(* CFC diagram, written out as Structured Text *)
(* KNX Master *)
KNX_master_2(I_Port := IoConfig_Globals.KNX_EIB_TP1_Interface_1, bPortKNX := 2);
STLV80_563.STLV80_A_563_KNX_Card_2_Status := KNX_master_2.sStatus = 'OK';
(* Rom 5H201 *)
(* RB601_V *)
(* RB601_HVAC *)
M2_001_5H201_RB601_V(bPortKNX := 2, dwIndex_DPT := 1, typDPT := typDPT);
STLV80_563.STLV80_A_563_5H201.RB601_V := M2_001_5H201_RB601_V.xSwitch_OUT;
M2_002_5H201_RB601_HVAC(bPortKNX := 2, dwIndex_DPT := 2, typDPT := typDPT);
STLV80_563.STLV80_A_563_5H201.RB601_HVAC := M2_002_5H201_RB601_HVAC.xSwitch_OUT;
(* RT601_CT *)
(* RY601_CV *)
M2_003_5H201_RT601_CT(bPortKNX := 2, dwIndex_DPT := 3, typDPT := typDPT);
STLV80_563.STLV80_A_563_5H201.RT601_CT := M2_003_5H201_RT601_CT.rValue_OUT;
M2_004_5H201_RY601_CV(bPortKNX := 2, dwIndex_DPT := 4, typDPT := typDPT);
STLV80_563.STLV80_A_563_5H201.RY601_CV := M2_004_5H201_RY601_CV.rValue_OUT;
(* LH601_OP *)
(* LH601_CMD *)
M2_005_5H201_LH601_OP(bPortKNX := 2, dwIndex_DPT := 5, rValue_IN := STLV80_563.STLV80_A_563_5H201.LH601_OP, xUpdate_KNX := i = 0, typDPT := typDPT);
M2_006_5H201_LH601_CMD(bPortKNX := 2, dwIndex_DPT := 6, xSwitch_IN := STLV80_563.STLV80_A_563_5H201.LH601_CMD, xUpdate_KNX := i = 1, typDPT := typDPT);
(* LC601_OP *)
(* LC601_CMD *)
M2_007_5H201_LC601_OP(bPortKNX := 2, dwIndex_DPT := 7, rValue_IN := STLV80_563.STLV80_A_563_5H201.LC601_OP, xUpdate_KNX := i = 2, typDPT := typDPT);
M2_008_5H201_LC601_CMD(bPortKNX := 2, dwIndex_DPT := 8, xSwitch_IN := STLV80_563.STLV80_A_563_5H201.LC601_CMD, xUpdate_KNX := i = 3, typDPT := typDPT);
(* RT601_SP *)
(* RT601_SP Feedback *)
M2_009_5H201_RT601_SP(bPortKNX := 2, dwIndex_DPT := 9, rValue_IN := STLV80_563.STLV80_A_563_5H201.RT601_SP_D, xUpdate_KNX := NOT STLV80_563.STLV80_A_563_5H201.RB601_HVAC, typDPT := typDPT);
M2_010_5H201_RT601_SP_FB(bPortKNX := 2, dwIndex_DPT := 10, typDPT := typDPT);
STLV80_563.STLV80_A_563_5H201.RT601_SP_IN := M2_010_5H201_RT601_SP_FB.rValue_OUT;
(* Rom 5I202 *)
(* RB601_V *)
(* RB601_HVAC *)
M2_011_5I202_RB601_V(bPortKNX := 2, dwIndex_DPT := 11, typDPT := typDPT);
STLV80_563.STLV80_A_563_5I202.RB601_V := M2_011_5I202_RB601_V.xSwitch_OUT;
M2_012_5I202_RB601_HVAC(bPortKNX := 2, dwIndex_DPT := 12, typDPT := typDPT);
STLV80_563.STLV80_A_563_5I202.RB601_HVAC := M2_012_5I202_RB601_HVAC.xSwitch_OUT;
(* RT601_CT *)
(* RY601_CV *)
M2_013_5I202_RT601_CT(bPortKNX := 2, dwIndex_DPT := 13, typDPT := typDPT);
STLV80_563.STLV80_A_563_5I202.RT601_CT := M2_013_5I202_RT601_CT.rValue_OUT;
M2_014_5I202_RY601_CV(bPortKNX := 2, dwIndex_DPT := 14, typDPT := typDPT);
STLV80_563.STLV80_A_563_5I202.RY601_CV := M2_014_5I202_RY601_CV.rValue_OUT;
(* LH601_OP *)
(* LH601_CMD *)
M2_015_5I202_LH601_OP(bPortKNX := 2, dwIndex_DPT := 15, rValue_IN := STLV80_563.STLV80_A_563_5I202.LH601_OP, xUpdate_KNX := i = 4, typDPT := typDPT);
M2_016_5I202_LH601_CMD(bPortKNX := 2, dwIndex_DPT := 16, xSwitch_IN := STLV80_563.STLV80_A_563_5I202.LH601_CMD, xUpdate_KNX := i = 5, typDPT := typDPT);
(* LC601_OP *)
(* LC601_CMD *)
M2_017_5I202_LC601_OP(bPortKNX := 2, dwIndex_DPT := 17, rValue_IN := STLV80_563.STLV80_A_563_5I202.LC601_OP, xUpdate_KNX := i = 6, typDPT := typDPT);
M2_018_5I202_LC601_CMD(bPortKNX := 2, dwIndex_DPT := 18, xSwitch_IN := STLV80_563.STLV80_A_563_5I202.LC601_CMD, xUpdate_KNX := i = 7, typDPT := typDPT);
(* RT601_SP *)
(* RT601_SP Feedback *)
M2_019_5I202_RT601_SP(bPortKNX := 2, dwIndex_DPT := 19, rValue_IN := STLV80_563.STLV80_A_563_5I202.RT601_SP_D, xUpdate_KNX := NOT STLV80_563.STLV80_A_563_5I202.RB601_HVAC, typDPT := typDPT);
M2_020_5I202_RT601_SP_FB(bPortKNX := 2, dwIndex_DPT := 20, typDPT := typDPT);
STLV80_563.STLV80_A_563_5I202.RT601_SP_IN := M2_020_5I202_RT601_SP_FB.rValue_OUT;
(* Rom 5I301 *)
(* RB601_V *)
(* RB601_HVAC *)
M2_021_5I301_RB601_V(bPortKNX := 2, dwIndex_DPT := 21, typDPT := typDPT);
STLV80_563.STLV80_A_563_5I301.RB601_V := M2_021_5I301_RB601_V.xSwitch_OUT;
M2_022_5I301_RB601_HVAC(bPortKNX := 2, dwIndex_DPT := 22, typDPT := typDPT);
STLV80_563.STLV80_A_563_5I301.RB601_HVAC := M2_022_5I301_RB601_HVAC.xSwitch_OUT;
(* RT601_CT *)
(* RY601_CV *)
M2_023_5I301_RT601_CT(bPortKNX := 2, dwIndex_DPT := 23, typDPT := typDPT);
STLV80_563.STLV80_A_563_5I301.RT601_CT := M2_023_5I301_RT601_CT.rValue_OUT;
M2_024_5I301_RY601_CV(bPortKNX := 2, dwIndex_DPT := 24, typDPT := typDPT);
STLV80_563.STLV80_A_563_5I301.RY601_CV := M2_024_5I301_RY601_CV.rValue_OUT;
(* LH601_OP *)
(* LH601_CMD *)
M2_025_5I301_LH601_OP(bPortKNX := 2, dwIndex_DPT := 25, rValue_IN := STLV80_563.STLV80_A_563_5I301.LH601_OP, xUpdate_KNX := i = 8, typDPT := typDPT);
M2_026_5I301_LH601_CMD(bPortKNX := 2, dwIndex_DPT := 26, xSwitch_IN := STLV80_563.STLV80_A_563_5I301.LH601_CMD, xUpdate_KNX := i = 9, typDPT := typDPT);
(* LC601_OP *)
(* LC601_CMD *)
M2_027_5I301_LC601_OP(bPortKNX := 2, dwIndex_DPT := 27, rValue_IN := STLV80_563.STLV80_A_563_5I301.LC601_OP, xUpdate_KNX := i = 10, typDPT := typDPT);
M2_028_5I301_LC601_CMD(bPortKNX := 2, dwIndex_DPT := 28, xSwitch_IN := STLV80_563.STLV80_A_563_5I301.LC601_CMD, xUpdate_KNX := i = 11, typDPT := typDPT);
(* RT601_SP *)
(* RT601_SP Feedback *)
M2_029_5I301_RT601_SP(bPortKNX := 2, dwIndex_DPT := 29, rValue_IN := STLV80_563.STLV80_A_563_5I301.RT601_SP_D, xUpdate_KNX := NOT STLV80_563.STLV80_A_563_5I301.RB601_HVAC, typDPT := typDPT);
M2_030_5I301_RT601_SP_FB(bPortKNX := 2, dwIndex_DPT := 30, typDPT := typDPT);
STLV80_563.STLV80_A_563_5I301.RT601_SP_IN := M2_030_5I301_RT601_SP_FB.rValue_OUT;
(* Rom 5I302 *)
(* RB601_V *)
(* RB601_HVAC *)
M2_031_5I302_RB601_V(bPortKNX := 2, dwIndex_DPT := 31, typDPT := typDPT);
STLV80_563.STLV80_A_563_5I302.RB601_V := M2_031_5I302_RB601_V.xSwitch_OUT;
M2_032_5I302_RB601_HVAC(bPortKNX := 2, dwIndex_DPT := 32, typDPT := typDPT);
STLV80_563.STLV80_A_563_5I302.RB601_HVAC := M2_032_5I302_RB601_HVAC.xSwitch_OUT;
(* RT601_CT *)
(* RY601_CV *)
M2_033_5I302_RT601_CT(bPortKNX := 2, dwIndex_DPT := 33, typDPT := typDPT);
STLV80_563.STLV80_A_563_5I302.RT601_CT := M2_033_5I302_RT601_CT.rValue_OUT;
M2_034_5I302_RY601_CV(bPortKNX := 2, dwIndex_DPT := 34, typDPT := typDPT);
STLV80_563.STLV80_A_563_5I302.RY601_CV := M2_034_5I302_RY601_CV.rValue_OUT;
(* LH601_OP *)
(* LH601_CMD *)
M2_035_5I302_LH601_OP(bPortKNX := 2, dwIndex_DPT := 35, rValue_IN := STLV80_563.STLV80_A_563_5I302.LH601_OP, xUpdate_KNX := i = 12, typDPT := typDPT);
M2_036_5I302_LH601_CMD(bPortKNX := 2, dwIndex_DPT := 36, xSwitch_IN := STLV80_563.STLV80_A_563_5I302.LH601_CMD, xUpdate_KNX := i = 13, typDPT := typDPT);
(* LC601_OP *)
(* LC601_CMD *)
M2_037_5I302_LC601_OP(bPortKNX := 2, dwIndex_DPT := 37, rValue_IN := STLV80_563.STLV80_A_563_5I302.LC601_OP, xUpdate_KNX := i = 14, typDPT := typDPT);
M2_038_5I302_LC601_CMD(bPortKNX := 2, dwIndex_DPT := 38, xSwitch_IN := STLV80_563.STLV80_A_563_5I302.LC601_CMD, xUpdate_KNX := i = 15, typDPT := typDPT);
(* RT601_SP *)
(* RT601_SP Feedback *)
M2_039_5I302_RT601_SP(bPortKNX := 2, dwIndex_DPT := 39, rValue_IN := STLV80_563.STLV80_A_563_5I302.RT601_SP_D, xUpdate_KNX := NOT STLV80_563.STLV80_A_563_5I302.RB601_HVAC, typDPT := typDPT);
M2_040_5I302_RT601_SP_FB(bPortKNX := 2, dwIndex_DPT := 40, typDPT := typDPT);
STLV80_563.STLV80_A_563_5I302.RT601_SP_IN := M2_040_5I302_RT601_SP_FB.rValue_OUT;
(* Rom 5J201 *)
(* RB601_V *)
(* RB601_HVAC *)
M2_041_5J201_RB601_V(bPortKNX := 2, dwIndex_DPT := 41, typDPT := typDPT);
STLV80_563.STLV80_A_563_5J201.RB601_V := M2_041_5J201_RB601_V.xSwitch_OUT;
M2_042_5J201_RB601_HVAC(bPortKNX := 2, dwIndex_DPT := 42, typDPT := typDPT);
STLV80_563.STLV80_A_563_5J201.RB601_HVAC := M2_042_5J201_RB601_HVAC.xSwitch_OUT;
(* RT601_CT *)
(* RY601_CV *)
M2_043_5J201_RT601_CT(bPortKNX := 2, dwIndex_DPT := 43, typDPT := typDPT);
STLV80_563.STLV80_A_563_5J201.RT601_CT := M2_043_5J201_RT601_CT.rValue_OUT;
M2_044_5J201_RY601_CV(bPortKNX := 2, dwIndex_DPT := 44, typDPT := typDPT);
STLV80_563.STLV80_A_563_5J201.RY601_CV := M2_044_5J201_RY601_CV.rValue_OUT;
(* LH601_OP *)
(* LH601_CMD *)
M2_045_5J201_LH601_OP(bPortKNX := 2, dwIndex_DPT := 45, rValue_IN := STLV80_563.STLV80_A_563_5J201.LH601_OP, xUpdate_KNX := i = 16, typDPT := typDPT);
M2_046_5J201_LH601_CMD(bPortKNX := 2, dwIndex_DPT := 46, xSwitch_IN := STLV80_563.STLV80_A_563_5J201.LH601_CMD, xUpdate_KNX := i = 17, typDPT := typDPT);
(* LC601_OP *)
(* LC601_CMD *)
M2_047_5J201_LC601_OP(bPortKNX := 2, dwIndex_DPT := 47, rValue_IN := STLV80_563.STLV80_A_563_5J201.LC601_OP, xUpdate_KNX := i = 18, typDPT := typDPT);
M2_048_5J201_LC601_CMD(bPortKNX := 2, dwIndex_DPT := 48, xSwitch_IN := STLV80_563.STLV80_A_563_5J201.LC601_CMD, xUpdate_KNX := i = 19, typDPT := typDPT);
(* RT601_SP *)
(* RT601_SP Feedback *)
M2_049_5J201_RT601_SP(bPortKNX := 2, dwIndex_DPT := 49, rValue_IN := STLV80_563.STLV80_A_563_5J201.RT601_SP_D, xUpdate_KNX := NOT STLV80_563.STLV80_A_563_5J201.RB601_HVAC, typDPT := typDPT);
M2_050_5J201_RT601_SP_FB(bPortKNX := 2, dwIndex_DPT := 50, typDPT := typDPT);
STLV80_563.STLV80_A_563_5J201.RT601_SP_IN := M2_050_5J201_RT601_SP_FB.rValue_OUT;
(* Rom 5J202 *)
(* RB601_V *)
(* RB601_HVAC *)
M2_051_5J202_RB601_V(bPortKNX := 2, dwIndex_DPT := 51, typDPT := typDPT);
STLV80_563.STLV80_A_563_5J202.RB601_V := M2_051_5J202_RB601_V.xSwitch_OUT;
M2_052_5J202_RB601_HVAC(bPortKNX := 2, dwIndex_DPT := 52, typDPT := typDPT);
STLV80_563.STLV80_A_563_5J202.RB601_HVAC := M2_052_5J202_RB601_HVAC.xSwitch_OUT;
(* RT601_CT *)
(* RY601_CV *)
M2_053_5J202_RT601_CT(bPortKNX := 2, dwIndex_DPT := 53, typDPT := typDPT);
STLV80_563.STLV80_A_563_5J202.RT601_CT := M2_053_5J202_RT601_CT.rValue_OUT;
M2_054_5J202_RY601_CV(bPortKNX := 2, dwIndex_DPT := 54, typDPT := typDPT);
STLV80_563.STLV80_A_563_5J202.RY601_CV := M2_054_5J202_RY601_CV.rValue_OUT;
(* LH601_OP *)
(* LH601_CMD *)
M2_055_5J202_LH601_OP(bPortKNX := 2, dwIndex_DPT := 55, rValue_IN := STLV80_563.STLV80_A_563_5J202.LH601_OP, xUpdate_KNX := i = 20, typDPT := typDPT);
M2_056_5J202_LH601_CMD(bPortKNX := 2, dwIndex_DPT := 56, xSwitch_IN := STLV80_563.STLV80_A_563_5J202.LH601_CMD, xUpdate_KNX := i = 21, typDPT := typDPT);
(* LC601_OP *)
(* LC601_CMD *)
M2_057_5J202_LC601_OP(bPortKNX := 2, dwIndex_DPT := 57, rValue_IN := STLV80_563.STLV80_A_563_5J202.LC601_OP, xUpdate_KNX := i = 22, typDPT := typDPT);
M2_058_5J202_LC601_CMD(bPortKNX := 2, dwIndex_DPT := 58, xSwitch_IN := STLV80_563.STLV80_A_563_5J202.LC601_CMD, xUpdate_KNX := i = 23, typDPT := typDPT);
(* RT601_SP *)
(* RT601_SP Feedback *)
M2_059_5J202_RT601_SP(bPortKNX := 2, dwIndex_DPT := 59, rValue_IN := STLV80_563.STLV80_A_563_5J202.RT601_SP_D, xUpdate_KNX := NOT STLV80_563.STLV80_A_563_5J202.RB601_HVAC, typDPT := typDPT);
M2_060_5J202_RT601_SP_FB(bPortKNX := 2, dwIndex_DPT := 60, typDPT := typDPT);
STLV80_563.STLV80_A_563_5J202.RT601_SP_IN := M2_060_5J202_RT601_SP_FB.rValue_OUT;
(* Rom 5J301 *)
(* RB601_V *)
(* RB601_HVAC *)
M2_061_5J301_RB601_V(bPortKNX := 2, dwIndex_DPT := 61, typDPT := typDPT);
STLV80_563.STLV80_A_563_5J301.RB601_V := M2_061_5J301_RB601_V.xSwitch_OUT;
M2_062_5J301_RB601_HVAC(bPortKNX := 2, dwIndex_DPT := 62, typDPT := typDPT);
STLV80_563.STLV80_A_563_5J301.RB601_HVAC := M2_062_5J301_RB601_HVAC.xSwitch_OUT;
(* RT601_CT *)
(* RY601_CV *)
M2_063_5J301_RT601_CT(bPortKNX := 2, dwIndex_DPT := 63, typDPT := typDPT);
STLV80_563.STLV80_A_563_5J301.RT601_CT := M2_063_5J301_RT601_CT.rValue_OUT;
M2_064_5J301_RY601_CV(bPortKNX := 2, dwIndex_DPT := 64, typDPT := typDPT);
STLV80_563.STLV80_A_563_5J301.RY601_CV := M2_064_5J301_RY601_CV.rValue_OUT;
(* LH601_OP *)
(* LH601_CMD *)
M2_065_5J301_LH601_OP(bPortKNX := 2, dwIndex_DPT := 65, rValue_IN := STLV80_563.STLV80_A_563_5J301.LH601_OP, xUpdate_KNX := i = 24, typDPT := typDPT);
M2_066_5J301_LH601_CMD(bPortKNX := 2, dwIndex_DPT := 66, xSwitch_IN := STLV80_563.STLV80_A_563_5J301.LH601_CMD, xUpdate_KNX := i = 25, typDPT := typDPT);
(* LC601_OP *)
(* LC601_CMD *)
M2_067_5J301_LC601_OP(bPortKNX := 2, dwIndex_DPT := 67, rValue_IN := STLV80_563.STLV80_A_563_5J301.LC601_OP, xUpdate_KNX := i = 26, typDPT := typDPT);
M2_068_5J301_LC601_CMD(bPortKNX := 2, dwIndex_DPT := 68, xSwitch_IN := STLV80_563.STLV80_A_563_5J301.LC601_CMD, xUpdate_KNX := i = 27, typDPT := typDPT);
(* RT601_SP *)
(* RT601_SP Feedback *)
M2_069_5J301_RT601_SP(bPortKNX := 2, dwIndex_DPT := 69, rValue_IN := STLV80_563.STLV80_A_563_5J301.RT601_SP_D, xUpdate_KNX := NOT STLV80_563.STLV80_A_563_5J301.RB601_HVAC, typDPT := typDPT);
M2_070_5J301_RT601_SP_FB(bPortKNX := 2, dwIndex_DPT := 70, typDPT := typDPT);
STLV80_563.STLV80_A_563_5J301.RT601_SP_IN := M2_070_5J301_RT601_SP_FB.rValue_OUT;
(* Rom 5K302 *)
(* RB601_V *)
(* RB601_HVAC *)
M2_071_5K302_RB601_V(bPortKNX := 2, dwIndex_DPT := 71, typDPT := typDPT);
STLV80_563.STLV80_A_563_5K302.RB601_V := M2_071_5K302_RB601_V.xSwitch_OUT;
M2_072_5K302_RB601_HVAC(bPortKNX := 2, dwIndex_DPT := 72, typDPT := typDPT);
STLV80_563.STLV80_A_563_5K302.RB601_HVAC := M2_072_5K302_RB601_HVAC.xSwitch_OUT;
(* RT601_CT *)
(* RY601_CV *)
M2_073_5K302_RT601_CT(bPortKNX := 2, dwIndex_DPT := 73, typDPT := typDPT);
STLV80_563.STLV80_A_563_5K302.RT601_CT := M2_073_5K302_RT601_CT.rValue_OUT;
M2_074_5K302_RY601_CV(bPortKNX := 2, dwIndex_DPT := 74, typDPT := typDPT);
STLV80_563.STLV80_A_563_5K302.RY601_CV := M2_074_5K302_RY601_CV.rValue_OUT;
(* LH601_OP *)
(* LH601_CMD *)
M2_075_5K302_LH601_OP(bPortKNX := 2, dwIndex_DPT := 75, rValue_IN := STLV80_563.STLV80_A_563_5K302.LH601_OP, xUpdate_KNX := i = 28, typDPT := typDPT);
M2_076_5K302_LH601_CMD(bPortKNX := 2, dwIndex_DPT := 76, xSwitch_IN := STLV80_563.STLV80_A_563_5K302.LH601_CMD, xUpdate_KNX := i = 29, typDPT := typDPT);
(* LC601_OP *)
(* LC601_CMD *)
M2_077_5K302_LC601_OP(bPortKNX := 2, dwIndex_DPT := 77, rValue_IN := STLV80_563.STLV80_A_563_5K302.LC601_OP, xUpdate_KNX := i = 30, typDPT := typDPT);
M2_078_5K302_LC601_CMD(bPortKNX := 2, dwIndex_DPT := 78, xSwitch_IN := STLV80_563.STLV80_A_563_5K302.LC601_CMD, xUpdate_KNX := i = 31, typDPT := typDPT);
(* RT601_SP *)
(* RT601_SP Feedback *)
M2_079_5K302_RT601_SP(bPortKNX := 2, dwIndex_DPT := 79, rValue_IN := STLV80_563.STLV80_A_563_5K302.RT601_SP_D, xUpdate_KNX := NOT STLV80_563.STLV80_A_563_5K302.RB601_HVAC, typDPT := typDPT);
M2_080_5K302_RT601_SP_FB(bPortKNX := 2, dwIndex_DPT := 80, typDPT := typDPT);
STLV80_563.STLV80_A_563_5K302.RT601_SP_IN := M2_080_5K302_RT601_SP_FB.rValue_OUT;
(* Rom 5K201 *)
(* RB601_V *)
(* RB601_HVAC *)
M2_081_5K201_RB601_V(bPortKNX := 2, dwIndex_DPT := 81, typDPT := typDPT);
STLV80_563.STLV80_A_563_5K201.RB601_V := M2_081_5K201_RB601_V.xSwitch_OUT;
M2_082_5K201_RB601_HVAC(bPortKNX := 2, dwIndex_DPT := 82, typDPT := typDPT);
STLV80_563.STLV80_A_563_5K201.RB601_HVAC := M2_082_5K201_RB601_HVAC.xSwitch_OUT;
(* RT601_CT *)
(* RY601_CV *)
M2_083_5K201_RT601_CT(bPortKNX := 2, dwIndex_DPT := 83, typDPT := typDPT);
STLV80_563.STLV80_A_563_5K201.RT601_CT := M2_083_5K201_RT601_CT.rValue_OUT;
M2_084_5K201_RY601_CV(bPortKNX := 2, dwIndex_DPT := 84, typDPT := typDPT);
STLV80_563.STLV80_A_563_5K201.RY601_CV := M2_084_5K201_RY601_CV.rValue_OUT;
(* LH601_OP *)
(* LH601_CMD *)
M2_085_5K201_LH601_OP(bPortKNX := 2, dwIndex_DPT := 85, rValue_IN := STLV80_563.STLV80_A_563_5K201.LH601_OP, xUpdate_KNX := i = 32, typDPT := typDPT);
M2_086_5K201_LH601_CMD(bPortKNX := 2, dwIndex_DPT := 86, xSwitch_IN := STLV80_563.STLV80_A_563_5K201.LH601_CMD, xUpdate_KNX := i = 33, typDPT := typDPT);
(* LC601_OP *)
(* LC601_CMD *)
M2_087_5K201_LC601_OP(bPortKNX := 2, dwIndex_DPT := 87, rValue_IN := STLV80_563.STLV80_A_563_5K201.LC601_OP, xUpdate_KNX := i = 34, typDPT := typDPT);
M2_088_5K201_LC601_CMD(bPortKNX := 2, dwIndex_DPT := 88, xSwitch_IN := STLV80_563.STLV80_A_563_5K201.LC601_CMD, xUpdate_KNX := i = 35, typDPT := typDPT);
(* RT601_SP *)
(* RT601_SP Feedback *)
M2_089_5K201_RT601_SP(bPortKNX := 2, dwIndex_DPT := 89, rValue_IN := STLV80_563.STLV80_A_563_5K201.RT601_SP_D, xUpdate_KNX := NOT STLV80_563.STLV80_A_563_5K201.RB601_HVAC, typDPT := typDPT);
M2_090_5K201_RT601_SP_FB(bPortKNX := 2, dwIndex_DPT := 90, typDPT := typDPT);
STLV80_563.STLV80_A_563_5K201.RT601_SP_IN := M2_090_5K201_RT601_SP_FB.rValue_OUT;
(* Rom 5K202 *)
(* RB601_V *)
(* RB601_HVAC *)
M2_091_5K202_RB601_V(bPortKNX := 2, dwIndex_DPT := 91, typDPT := typDPT);
STLV80_563.STLV80_A_563_5K202.RB601_V := M2_091_5K202_RB601_V.xSwitch_OUT;
M2_092_5K202_RB601_HVAC(bPortKNX := 2, dwIndex_DPT := 92, typDPT := typDPT);
STLV80_563.STLV80_A_563_5K202.RB601_HVAC := M2_092_5K202_RB601_HVAC.xSwitch_OUT;
(* RT601_CT *)
(* RY601_CV *)
M2_093_5K202_RT601_CT(bPortKNX := 2, dwIndex_DPT := 93, typDPT := typDPT);
STLV80_563.STLV80_A_563_5K202.RT601_CT := M2_093_5K202_RT601_CT.rValue_OUT;
M2_094_5K202_RY601_CV(bPortKNX := 2, dwIndex_DPT := 94, typDPT := typDPT);
STLV80_563.STLV80_A_563_5K202.RY601_CV := M2_094_5K202_RY601_CV.rValue_OUT;
(* LH601_OP *)
(* LH601_CMD *)
M2_095_5K202_LH601_OP(bPortKNX := 2, dwIndex_DPT := 95, rValue_IN := STLV80_563.STLV80_A_563_5K202.LH601_OP, xUpdate_KNX := i = 36, typDPT := typDPT);
M2_096_5K202_LH601_CMD(bPortKNX := 2, dwIndex_DPT := 96, xSwitch_IN := STLV80_563.STLV80_A_563_5K202.LH601_CMD, xUpdate_KNX := i = 37, typDPT := typDPT);
(* LC601_OP *)
(* LC601_CMD *)
M2_097_5K202_LC601_OP(bPortKNX := 2, dwIndex_DPT := 97, rValue_IN := STLV80_563.STLV80_A_563_5K202.LC601_OP, xUpdate_KNX := i = 38, typDPT := typDPT);
M2_098_5K202_LC601_CMD(bPortKNX := 2, dwIndex_DPT := 98, xSwitch_IN := STLV80_563.STLV80_A_563_5K202.LC601_CMD, xUpdate_KNX := i = 39, typDPT := typDPT);
(* RT601_SP *)
(* RT601_SP Feedback *)
M2_099_5K202_RT601_SP(bPortKNX := 2, dwIndex_DPT := 99, rValue_IN := STLV80_563.STLV80_A_563_5K202.RT601_SP_D, xUpdate_KNX := NOT STLV80_563.STLV80_A_563_5K202.RB601_HVAC, typDPT := typDPT);
M2_100_5K202_RT601_SP_FB(bPortKNX := 2, dwIndex_DPT := 100, typDPT := typDPT);
STLV80_563.STLV80_A_563_5K202.RT601_SP_IN := M2_100_5K202_RT601_SP_FB.rValue_OUT;
(* Rom 5K301 *)
(* RB601_V *)
(* RB601_HVAC *)
M2_101_5K301_RB601_V(bPortKNX := 2, dwIndex_DPT := 101, typDPT := typDPT);
STLV80_563.STLV80_A_563_5K301.RB601_V := M2_101_5K301_RB601_V.xSwitch_OUT;
M2_102_5K301_RB601_HVAC(bPortKNX := 2, dwIndex_DPT := 102, typDPT := typDPT);
STLV80_563.STLV80_A_563_5K301.RB601_HVAC := M2_102_5K301_RB601_HVAC.xSwitch_OUT;
(* RT601_CT *)
(* RY601_CV *)
M2_103_5K301_RT601_CT(bPortKNX := 2, dwIndex_DPT := 103, typDPT := typDPT);
STLV80_563.STLV80_A_563_5K301.RT601_CT := M2_103_5K301_RT601_CT.rValue_OUT;
M2_104_5K301_RY601_CV(bPortKNX := 2, dwIndex_DPT := 104, typDPT := typDPT);
STLV80_563.STLV80_A_563_5K301.RY601_CV := M2_104_5K301_RY601_CV.rValue_OUT;
(* LH601_OP *)
(* LH601_CMD *)
M2_105_5K301_LH601_OP(bPortKNX := 2, dwIndex_DPT := 105, rValue_IN := STLV80_563.STLV80_A_563_5K301.LH601_OP, xUpdate_KNX := i = 40, typDPT := typDPT);
M2_106_5K301_LH601_CMD(bPortKNX := 2, dwIndex_DPT := 106, xSwitch_IN := STLV80_563.STLV80_A_563_5K301.LH601_CMD, xUpdate_KNX := i = 41, typDPT := typDPT);
(* LC601_OP *)
(* LC601_CMD *)
M2_107_5K301_LC601_OP(bPortKNX := 2, dwIndex_DPT := 107, rValue_IN := STLV80_563.STLV80_A_563_5K301.LC601_OP, xUpdate_KNX := i = 42, typDPT := typDPT);
M2_108_5K301_LC601_CMD(bPortKNX := 2, dwIndex_DPT := 108, xSwitch_IN := STLV80_563.STLV80_A_563_5K301.LC601_CMD, xUpdate_KNX := i = 43, typDPT := typDPT);
(* RT601_SP *)
(* RT601_SP Feedback *)
M2_109_5K301_RT601_SP(bPortKNX := 2, dwIndex_DPT := 109, rValue_IN := STLV80_563.STLV80_A_563_5K301.RT601_SP_D, xUpdate_KNX := NOT STLV80_563.STLV80_A_563_5K301.RB601_HVAC, typDPT := typDPT);
M2_110_5K301_RT601_SP_FB(bPortKNX := 2, dwIndex_DPT := 110, typDPT := typDPT);
STLV80_563.STLV80_A_563_5K301.RT601_SP_IN := M2_110_5K301_RT601_SP_FB.rValue_OUT;
(* Rom 5L201 *)
(* RB601_V *)
(* RB601_HVAC *)
M2_111_5L201_RB601_V(bPortKNX := 2, dwIndex_DPT := 111, typDPT := typDPT);
STLV80_563.STLV80_A_563_5L201.RB601_V := M2_111_5L201_RB601_V.xSwitch_OUT;
M2_112_5L201_RB601_HVAC(bPortKNX := 2, dwIndex_DPT := 112, typDPT := typDPT);
STLV80_563.STLV80_A_563_5L201.RB601_HVAC := M2_112_5L201_RB601_HVAC.xSwitch_OUT;
(* RT601_CT *)
(* RY601_CV *)
M2_113_5L201_RT601_CT(bPortKNX := 2, dwIndex_DPT := 113, typDPT := typDPT);
STLV80_563.STLV80_A_563_5L201.RT601_CT := M2_113_5L201_RT601_CT.rValue_OUT;
M2_114_5L201_RY601_CV(bPortKNX := 2, dwIndex_DPT := 114, typDPT := typDPT);
STLV80_563.STLV80_A_563_5L201.RY601_CV := M2_114_5L201_RY601_CV.rValue_OUT;
(* LH601_OP *)
(* LH601_CMD *)
M2_115_5L201_LH601_OP(bPortKNX := 2, dwIndex_DPT := 115, rValue_IN := STLV80_563.STLV80_A_563_5L201.LH601_OP, xUpdate_KNX := i = 44, typDPT := typDPT);
M2_116_5L201_LH601_CMD(bPortKNX := 2, dwIndex_DPT := 116, xSwitch_IN := STLV80_563.STLV80_A_563_5L201.LH601_CMD, xUpdate_KNX := i = 45, typDPT := typDPT);
(* LC601_OP *)
(* LC601_CMD *)
M2_117_5L201_LC601_OP(bPortKNX := 2, dwIndex_DPT := 117, rValue_IN := STLV80_563.STLV80_A_563_5L201.LC601_OP, xUpdate_KNX := i = 46, typDPT := typDPT);
M2_118_5L201_LC601_CMD(bPortKNX := 2, dwIndex_DPT := 118, xSwitch_IN := STLV80_563.STLV80_A_563_5L201.LC601_CMD, xUpdate_KNX := i = 47, typDPT := typDPT);
(* RT601_SP *)
(* RT601_SP Feedback *)
M2_119_5L201_RT601_SP(bPortKNX := 2, dwIndex_DPT := 119, rValue_IN := STLV80_563.STLV80_A_563_5L201.RT601_SP_D, xUpdate_KNX := NOT STLV80_563.STLV80_A_563_5L201.RB601_HVAC, typDPT := typDPT);
M2_120_5L201_RT601_SP_FB(bPortKNX := 2, dwIndex_DPT := 120, typDPT := typDPT);
STLV80_563.STLV80_A_563_5L201.RT601_SP_IN := M2_120_5L201_RT601_SP_FB.rValue_OUT;
(* Rom 5L202 *)
(* RB601_V *)
(* RB601_HVAC *)
M2_121_5L202_RB601_V(bPortKNX := 2, dwIndex_DPT := 121, typDPT := typDPT);
STLV80_563.STLV80_A_563_5L202.RB601_V := M2_121_5L202_RB601_V.xSwitch_OUT;
M2_122_5L202_RB601_HVAC(bPortKNX := 2, dwIndex_DPT := 122, typDPT := typDPT);
STLV80_563.STLV80_A_563_5L202.RB601_HVAC := M2_122_5L202_RB601_HVAC.xSwitch_OUT;
(* RT601_CT *)
(* RY601_CV *)
M2_123_5L202_RT601_CT(bPortKNX := 2, dwIndex_DPT := 123, typDPT := typDPT);
STLV80_563.STLV80_A_563_5L202.RT601_CT := M2_123_5L202_RT601_CT.rValue_OUT;
M2_124_5L202_RY601_CV(bPortKNX := 2, dwIndex_DPT := 124, typDPT := typDPT);
STLV80_563.STLV80_A_563_5L202.RY601_CV := M2_124_5L202_RY601_CV.rValue_OUT;
(* LH601_OP *)
(* LH601_CMD *)
M2_125_5L202_LH601_OP(bPortKNX := 2, dwIndex_DPT := 125, rValue_IN := STLV80_563.STLV80_A_563_5L202.LH601_OP, xUpdate_KNX := i = 48, typDPT := typDPT);
M2_126_5L202_LH601_CMD(bPortKNX := 2, dwIndex_DPT := 126, xSwitch_IN := STLV80_563.STLV80_A_563_5L202.LH601_CMD, xUpdate_KNX := i = 49, typDPT := typDPT);
(* LC601_OP *)
(* LC601_CMD *)
M2_127_5L202_LC601_OP(bPortKNX := 2, dwIndex_DPT := 127, rValue_IN := STLV80_563.STLV80_A_563_5L202.LC601_OP, xUpdate_KNX := i = 50, typDPT := typDPT);
M2_128_5L202_LC601_CMD(bPortKNX := 2, dwIndex_DPT := 128, xSwitch_IN := STLV80_563.STLV80_A_563_5L202.LC601_CMD, xUpdate_KNX := i = 51, typDPT := typDPT);
(* RT601_SP *)
(* RT601_SP Feedback *)
M2_129_5L202_RT601_SP(bPortKNX := 2, dwIndex_DPT := 129, rValue_IN := STLV80_563.STLV80_A_563_5L202.RT601_SP_D, xUpdate_KNX := NOT STLV80_563.STLV80_A_563_5L202.RB601_HVAC, typDPT := typDPT);
M2_130_5L202_RT601_SP_FB(bPortKNX := 2, dwIndex_DPT := 130, typDPT := typDPT);
STLV80_563.STLV80_A_563_5L202.RT601_SP_IN := M2_130_5L202_RT601_SP_FB.rValue_OUT;
(* Rom 5L301 *)
(* RB601_V *)
(* RB601_HVAC *)
M2_131_5L301_RB601_V(bPortKNX := 2, dwIndex_DPT := 131, typDPT := typDPT);
STLV80_563.STLV80_A_563_5L301.RB601_V := M2_131_5L301_RB601_V.xSwitch_OUT;
M2_132_5L301_RB601_HVAC(bPortKNX := 2, dwIndex_DPT := 132, typDPT := typDPT);
STLV80_563.STLV80_A_563_5L301.RB601_HVAC := M2_132_5L301_RB601_HVAC.xSwitch_OUT;
(* RT601_CT *)
(* RY601_CV *)
M2_133_5L301_RT601_CT(bPortKNX := 2, dwIndex_DPT := 133, typDPT := typDPT);
STLV80_563.STLV80_A_563_5L301.RT601_CT := M2_133_5L301_RT601_CT.rValue_OUT;
M2_134_5L301_RY601_CV(bPortKNX := 2, dwIndex_DPT := 134, typDPT := typDPT);
STLV80_563.STLV80_A_563_5L301.RY601_CV := M2_134_5L301_RY601_CV.rValue_OUT;
(* LH601_OP *)
(* LH601_CMD *)
M2_135_5L301_LH601_OP(bPortKNX := 2, dwIndex_DPT := 135, rValue_IN := STLV80_563.STLV80_A_563_5L301.LH601_OP, xUpdate_KNX := i = 52, typDPT := typDPT);
M2_136_5L301_LH601_CMD(bPortKNX := 2, dwIndex_DPT := 136, xSwitch_IN := STLV80_563.STLV80_A_563_5L301.LH601_CMD, xUpdate_KNX := i = 53, typDPT := typDPT);
(* LC601_OP *)
(* LC601_CMD *)
M2_137_5L301_LC601_OP(bPortKNX := 2, dwIndex_DPT := 137, rValue_IN := STLV80_563.STLV80_A_563_5L301.LC601_OP, xUpdate_KNX := i = 54, typDPT := typDPT);
M2_138_5L301_LC601_CMD(bPortKNX := 2, dwIndex_DPT := 138, xSwitch_IN := STLV80_563.STLV80_A_563_5L301.LC601_CMD, xUpdate_KNX := i = 55, typDPT := typDPT);
(* RT601_SP *)
(* RT601_SP Feedback *)
M2_139_5L301_RT601_SP(bPortKNX := 2, dwIndex_DPT := 139, rValue_IN := STLV80_563.STLV80_A_563_5L301.RT601_SP_D, xUpdate_KNX := NOT STLV80_563.STLV80_A_563_5L301.RB601_HVAC, typDPT := typDPT);
M2_140_5L301_RT601_SP_FB(bPortKNX := 2, dwIndex_DPT := 140, typDPT := typDPT);
STLV80_563.STLV80_A_563_5L301.RT601_SP_IN := M2_140_5L301_RT601_SP_FB.rValue_OUT;
(* Rom 5L302 *)
(* RB601_V *)
(* RB601_HVAC *)
M2_141_5L302_RB601_V(bPortKNX := 2, dwIndex_DPT := 141, typDPT := typDPT);
STLV80_563.STLV80_A_563_5L302.RB601_V := M2_141_5L302_RB601_V.xSwitch_OUT;
M2_142_5L302_RB601_HVAC(bPortKNX := 2, dwIndex_DPT := 142, typDPT := typDPT);
STLV80_563.STLV80_A_563_5L302.RB601_HVAC := M2_142_5L302_RB601_HVAC.xSwitch_OUT;
(* RT601_CT *)
(* RY601_CV *)
M2_143_5L302_RT601_CT(bPortKNX := 2, dwIndex_DPT := 143, typDPT := typDPT);
STLV80_563.STLV80_A_563_5L302.RT601_CT := M2_143_5L302_RT601_CT.rValue_OUT;
M2_144_5L302_RY601_CV(bPortKNX := 2, dwIndex_DPT := 144, typDPT := typDPT);
STLV80_563.STLV80_A_563_5L302.RY601_CV := M2_144_5L302_RY601_CV.rValue_OUT;
(* LH601_OP *)
(* LH601_CMD *)
M2_145_5L302_LH601_OP(bPortKNX := 2, dwIndex_DPT := 145, rValue_IN := STLV80_563.STLV80_A_563_5L302.LH601_OP, xUpdate_KNX := i = 56, typDPT := typDPT);
M2_146_5L302_LH601_CMD(bPortKNX := 2, dwIndex_DPT := 146, xSwitch_IN := STLV80_563.STLV80_A_563_5L302.LH601_CMD, xUpdate_KNX := i = 57, typDPT := typDPT);
(* LC601_OP *)
(* LC601_CMD *)
M2_147_5L302_LC601_OP(bPortKNX := 2, dwIndex_DPT := 147, rValue_IN := STLV80_563.STLV80_A_563_5L302.LC601_OP, xUpdate_KNX := i = 58, typDPT := typDPT);
M2_148_5L302_LC601_CMD(bPortKNX := 2, dwIndex_DPT := 148, xSwitch_IN := STLV80_563.STLV80_A_563_5L302.LC601_CMD, xUpdate_KNX := i = 59, typDPT := typDPT);
(* RT601_SP *)
(* RT601_SP Feedback *)
M2_149_5L302_RT601_SP(bPortKNX := 2, dwIndex_DPT := 149, rValue_IN := STLV80_563.STLV80_A_563_5L302.RT601_SP_D, xUpdate_KNX := NOT STLV80_563.STLV80_A_563_5L302.RB601_HVAC, typDPT := typDPT);
M2_150_5L302_RT601_SP_FB(bPortKNX := 2, dwIndex_DPT := 150, typDPT := typDPT);
STLV80_563.STLV80_A_563_5L302.RT601_SP_IN := M2_150_5L302_RT601_SP_FB.rValue_OUT;
(* Rom 5M201 *)
(* RB601_V *)
(* RB601_HVAC *)
M2_151_5M201_RB601_V(bPortKNX := 2, dwIndex_DPT := 151, typDPT := typDPT);
STLV80_563.STLV80_A_563_5M201.RB601_V := M2_151_5M201_RB601_V.xSwitch_OUT;
M2_152_5M201_RB601_HVAC(bPortKNX := 2, dwIndex_DPT := 152, typDPT := typDPT);
STLV80_563.STLV80_A_563_5M201.RB601_HVAC := M2_152_5M201_RB601_HVAC.xSwitch_OUT;
(* RT601_CT *)
(* RY601_CV *)
M2_153_5M201_RT601_CT(bPortKNX := 2, dwIndex_DPT := 153, typDPT := typDPT);
STLV80_563.STLV80_A_563_5M201.RT601_CT := M2_153_5M201_RT601_CT.rValue_OUT;
M2_154_5M201_RY601_CV(bPortKNX := 2, dwIndex_DPT := 154, typDPT := typDPT);
STLV80_563.STLV80_A_563_5M201.RY601_CV := M2_154_5M201_RY601_CV.rValue_OUT;
(* LH601_OP *)
(* LH601_CMD *)
M2_155_5M201_LH601_OP(bPortKNX := 2, dwIndex_DPT := 155, rValue_IN := STLV80_563.STLV80_A_563_5M201.LH601_OP, xUpdate_KNX := i = 60, typDPT := typDPT);
M2_156_5M201_LH601_CMD(bPortKNX := 2, dwIndex_DPT := 156, xSwitch_IN := STLV80_563.STLV80_A_563_5M201.LH601_CMD, xUpdate_KNX := i = 61, typDPT := typDPT);
(* LC601_OP *)
(* LC601_CMD *)
M2_157_5M201_LC601_OP(bPortKNX := 2, dwIndex_DPT := 157, rValue_IN := STLV80_563.STLV80_A_563_5M201.LC601_OP, xUpdate_KNX := i = 62, typDPT := typDPT);
M2_158_5M201_LC601_CMD(bPortKNX := 2, dwIndex_DPT := 158, xSwitch_IN := STLV80_563.STLV80_A_563_5M201.LC601_CMD, xUpdate_KNX := i = 63, typDPT := typDPT);
(* RT601_SP *)
(* RT601_SP Feedback *)
M2_159_5M201_RT601_SP(bPortKNX := 2, dwIndex_DPT := 159, rValue_IN := STLV80_563.STLV80_A_563_5M201.RT601_SP_D, xUpdate_KNX := NOT STLV80_563.STLV80_A_563_5M201.RB601_HVAC, typDPT := typDPT);
M2_160_5M201_RT601_SP_FB(bPortKNX := 2, dwIndex_DPT := 160, typDPT := typDPT);
STLV80_563.STLV80_A_563_5M201.RT601_SP_IN := M2_160_5M201_RT601_SP_FB.rValue_OUT;
(* Rom 5M202 *)
(* RB601_V *)
(* RB601_HVAC *)
M2_161_5M202_RB601_V(bPortKNX := 2, dwIndex_DPT := 161, typDPT := typDPT);
STLV80_563.STLV80_A_563_5M202.RB601_V := M2_161_5M202_RB601_V.xSwitch_OUT;
M2_162_5M202_RB601_HVAC(bPortKNX := 2, dwIndex_DPT := 162, typDPT := typDPT);
STLV80_563.STLV80_A_563_5M202.RB601_HVAC := M2_162_5M202_RB601_HVAC.xSwitch_OUT;
(* RT601_CT *)
(* RY601_CV *)
M2_163_5M202_RT601_CT(bPortKNX := 2, dwIndex_DPT := 163, typDPT := typDPT);
STLV80_563.STLV80_A_563_5M202.RT601_CT := M2_163_5M202_RT601_CT.rValue_OUT;
M2_164_5M202_RY601_CV(bPortKNX := 2, dwIndex_DPT := 164, typDPT := typDPT);
STLV80_563.STLV80_A_563_5M202.RY601_CV := M2_164_5M202_RY601_CV.rValue_OUT;
(* LH601_OP *)
(* LH601_CMD *)
M2_165_5M202_LH601_OP(bPortKNX := 2, dwIndex_DPT := 165, rValue_IN := STLV80_563.STLV80_A_563_5M202.LH601_OP, xUpdate_KNX := i = 64, typDPT := typDPT);
M2_166_5M202_LH601_CMD(bPortKNX := 2, dwIndex_DPT := 166, xSwitch_IN := STLV80_563.STLV80_A_563_5M202.LH601_CMD, xUpdate_KNX := i = 65, typDPT := typDPT);
(* LC601_OP *)
(* LC601_CMD *)
M2_167_5M202_LC601_OP(bPortKNX := 2, dwIndex_DPT := 167, rValue_IN := STLV80_563.STLV80_A_563_5M202.LC601_OP, xUpdate_KNX := i = 66, typDPT := typDPT);
M2_168_5M202_LC601_CMD(bPortKNX := 2, dwIndex_DPT := 168, xSwitch_IN := STLV80_563.STLV80_A_563_5M202.LC601_CMD, xUpdate_KNX := i = 67, typDPT := typDPT);
(* RT601_SP *)
(* RT601_SP Feedback *)
M2_169_5M202_RT601_SP(bPortKNX := 2, dwIndex_DPT := 169, rValue_IN := STLV80_563.STLV80_A_563_5M202.RT601_SP_D, xUpdate_KNX := NOT STLV80_563.STLV80_A_563_5M202.RB601_HVAC, typDPT := typDPT);
M2_170_5M202_RT601_SP_FB(bPortKNX := 2, dwIndex_DPT := 170, typDPT := typDPT);
STLV80_563.STLV80_A_563_5M202.RT601_SP_IN := M2_170_5M202_RT601_SP_FB.rValue_OUT;
(* Rom 5M301 *)
(* RB601_V *)
(* RB601_HVAC *)
M2_171_5M301_RB601_V(bPortKNX := 2, dwIndex_DPT := 171, typDPT := typDPT);
STLV80_563.STLV80_A_563_5M301.RB601_V := M2_171_5M301_RB601_V.xSwitch_OUT;
M2_172_5M301_RB601_HVAC(bPortKNX := 2, dwIndex_DPT := 172, typDPT := typDPT);
STLV80_563.STLV80_A_563_5M301.RB601_HVAC := M2_172_5M301_RB601_HVAC.xSwitch_OUT;
(* RT601_CT *)
(* RY601_CV *)
M2_173_5M301_RT601_CT(bPortKNX := 2, dwIndex_DPT := 173, typDPT := typDPT);
STLV80_563.STLV80_A_563_5M301.RT601_CT := M2_173_5M301_RT601_CT.rValue_OUT;
M2_174_5M301_RY601_CV(bPortKNX := 2, dwIndex_DPT := 174, typDPT := typDPT);
STLV80_563.STLV80_A_563_5M301.RY601_CV := M2_174_5M301_RY601_CV.rValue_OUT;
(* LH601_OP *)
(* LH601_CMD *)
M2_175_5M301_LH601_OP(bPortKNX := 2, dwIndex_DPT := 175, rValue_IN := STLV80_563.STLV80_A_563_5M301.LH601_OP, xUpdate_KNX := i = 68, typDPT := typDPT);
M2_176_5M301_LH601_CMD(bPortKNX := 2, dwIndex_DPT := 176, xSwitch_IN := STLV80_563.STLV80_A_563_5M301.LH601_CMD, xUpdate_KNX := i = 69, typDPT := typDPT);
(* LC601_OP *)
(* LC601_CMD *)
M2_177_5M301_LC601_OP(bPortKNX := 2, dwIndex_DPT := 177, rValue_IN := STLV80_563.STLV80_A_563_5M301.LC601_OP, xUpdate_KNX := i = 70, typDPT := typDPT);
M2_178_5M301_LC601_CMD(bPortKNX := 2, dwIndex_DPT := 178, xSwitch_IN := STLV80_563.STLV80_A_563_5M301.LC601_CMD, xUpdate_KNX := i = 71, typDPT := typDPT);
(* RT601_SP *)
(* RT601_SP Feedback *)
M2_179_5M301_RT601_SP(bPortKNX := 2, dwIndex_DPT := 179, rValue_IN := STLV80_563.STLV80_A_563_5M301.RT601_SP_D, xUpdate_KNX := NOT STLV80_563.STLV80_A_563_5M301.RB601_HVAC, typDPT := typDPT);
M2_180_5M301_RT601_SP_FB(bPortKNX := 2, dwIndex_DPT := 180, typDPT := typDPT);
STLV80_563.STLV80_A_563_5M301.RT601_SP_IN := M2_180_5M301_RT601_SP_FB.rValue_OUT;
(* Rom 5N201 *)
(* RB601_V *)
(* RB601_HVAC *)
M2_181_5N201_RB601_V(bPortKNX := 2, dwIndex_DPT := 181, typDPT := typDPT);
STLV80_563.STLV80_A_563_5N201.RB601_V := M2_181_5N201_RB601_V.xSwitch_OUT;
M2_182_5N201_RB601_HVAC(bPortKNX := 2, dwIndex_DPT := 182, typDPT := typDPT);
STLV80_563.STLV80_A_563_5N201.RB601_HVAC := M2_182_5N201_RB601_HVAC.xSwitch_OUT;
(* RT601_CT *)
(* RY601_CV *)
M2_183_5N201_RT601_CT(bPortKNX := 2, dwIndex_DPT := 183, typDPT := typDPT);
STLV80_563.STLV80_A_563_5N201.RT601_CT := M2_183_5N201_RT601_CT.rValue_OUT;
M2_184_5N201_RY601_CV(bPortKNX := 2, dwIndex_DPT := 184, typDPT := typDPT);
STLV80_563.STLV80_A_563_5N201.RY601_CV := M2_184_5N201_RY601_CV.rValue_OUT;
(* LH601_OP *)
(* LH601_CMD *)
M2_185_5N201_LH601_OP(bPortKNX := 2, dwIndex_DPT := 185, rValue_IN := STLV80_563.STLV80_A_563_5N201.LH601_OP, xUpdate_KNX := i = 72, typDPT := typDPT);
M2_186_5N201_LH601_CMD(bPortKNX := 2, dwIndex_DPT := 186, xSwitch_IN := STLV80_563.STLV80_A_563_5N201.LH601_CMD, xUpdate_KNX := i = 73, typDPT := typDPT);
(* LC601_OP *)
(* LC601_CMD *)
M2_187_5N201_LC601_OP(bPortKNX := 2, dwIndex_DPT := 187, rValue_IN := STLV80_563.STLV80_A_563_5N201.LC601_OP, xUpdate_KNX := i = 74, typDPT := typDPT);
M2_188_5N201_LC601_CMD(bPortKNX := 2, dwIndex_DPT := 188, xSwitch_IN := STLV80_563.STLV80_A_563_5N201.LC601_CMD, xUpdate_KNX := i = 75, typDPT := typDPT);
(* RT601_SP *)
(* RT601_SP Feedback *)
M2_189_5N201_RT601_SP(bPortKNX := 2, dwIndex_DPT := 189, rValue_IN := STLV80_563.STLV80_A_563_5N201.RT601_SP_D, xUpdate_KNX := NOT STLV80_563.STLV80_A_563_5N201.RB601_HVAC, typDPT := typDPT);
M2_190_5N201_RT601_SP_FB(bPortKNX := 2, dwIndex_DPT := 190, typDPT := typDPT);
STLV80_563.STLV80_A_563_5N201.RT601_SP_IN := M2_190_5N201_RT601_SP_FB.rValue_OUT;
(* Rom 5N202 *)
(* RB601_V *)
(* RB601_HVAC *)
M2_191_5N202_RB601_V(bPortKNX := 2, dwIndex_DPT := 191, typDPT := typDPT);
STLV80_563.STLV80_A_563_5N202.RB601_V := M2_191_5N202_RB601_V.xSwitch_OUT;
M2_192_5N202_RB601_HVAC(bPortKNX := 2, dwIndex_DPT := 192, typDPT := typDPT);
STLV80_563.STLV80_A_563_5N202.RB601_HVAC := M2_192_5N202_RB601_HVAC.xSwitch_OUT;
(* RT601_CT *)
(* RY601_CV *)
M2_193_5N202_RT601_CT(bPortKNX := 2, dwIndex_DPT := 193, typDPT := typDPT);
STLV80_563.STLV80_A_563_5N202.RT601_CT := M2_193_5N202_RT601_CT.rValue_OUT;
M2_194_5N202_RY601_CV(bPortKNX := 2, dwIndex_DPT := 194, typDPT := typDPT);
STLV80_563.STLV80_A_563_5N202.RY601_CV := M2_194_5N202_RY601_CV.rValue_OUT;
(* LH601_OP *)
(* LH601_CMD *)
M2_195_5N202_LH601_OP(bPortKNX := 2, dwIndex_DPT := 195, rValue_IN := STLV80_563.STLV80_A_563_5N202.LH601_OP, xUpdate_KNX := i = 76, typDPT := typDPT);
M2_196_5N202_LH601_CMD(bPortKNX := 2, dwIndex_DPT := 196, xSwitch_IN := STLV80_563.STLV80_A_563_5N202.LH601_CMD, xUpdate_KNX := i = 77, typDPT := typDPT);
(* LC601_OP *)
(* LC601_CMD *)
M2_197_5N202_LC601_OP(bPortKNX := 2, dwIndex_DPT := 197, rValue_IN := STLV80_563.STLV80_A_563_5N202.LC601_OP, xUpdate_KNX := i = 78, typDPT := typDPT);
M2_198_5N202_LC601_CMD(bPortKNX := 2, dwIndex_DPT := 198, xSwitch_IN := STLV80_563.STLV80_A_563_5N202.LC601_CMD, xUpdate_KNX := i = 79, typDPT := typDPT);
(* RT601_SP *)
(* RT601_SP Feedback *)
M2_199_5N202_RT601_SP(bPortKNX := 2, dwIndex_DPT := 199, rValue_IN := STLV80_563.STLV80_A_563_5N202.RT601_SP_D, xUpdate_KNX := NOT STLV80_563.STLV80_A_563_5N202.RB601_HVAC, typDPT := typDPT);
M2_200_5N202_RT601_SP_FB(bPortKNX := 2, dwIndex_DPT := 200, typDPT := typDPT);
STLV80_563.STLV80_A_563_5N202.RT601_SP_IN := M2_200_5N202_RT601_SP_FB.rValue_OUT;
(* Rom 5N301 *)
(* RB601_V *)
(* RB601_HVAC *)
M2_201_5N301_RB601_V(bPortKNX := 2, dwIndex_DPT := 201, typDPT := typDPT);
STLV80_563.STLV80_A_563_5N301.RB601_V := M2_201_5N301_RB601_V.xSwitch_OUT;
M2_202_5N301_RB601_HVAC(bPortKNX := 2, dwIndex_DPT := 202, typDPT := typDPT);
STLV80_563.STLV80_A_563_5N301.RB601_HVAC := M2_202_5N301_RB601_HVAC.xSwitch_OUT;
(* RT601_CT *)
(* RY601_CV *)
M2_203_5N301_RT601_CT(bPortKNX := 2, dwIndex_DPT := 203, typDPT := typDPT);
STLV80_563.STLV80_A_563_5N301.RT601_CT := M2_203_5N301_RT601_CT.rValue_OUT;
M2_204_5N301_RY601_CV(bPortKNX := 2, dwIndex_DPT := 204, typDPT := typDPT);
STLV80_563.STLV80_A_563_5N301.RY601_CV := M2_204_5N301_RY601_CV.rValue_OUT;
(* LH601_OP *)
(* LH601_CMD *)
M2_205_5N301_LH601_OP(bPortKNX := 2, dwIndex_DPT := 205, rValue_IN := STLV80_563.STLV80_A_563_5N301.LH601_OP, xUpdate_KNX := i = 80, typDPT := typDPT);
M2_206_5N301_LH601_CMD(bPortKNX := 2, dwIndex_DPT := 206, xSwitch_IN := STLV80_563.STLV80_A_563_5N301.LH601_CMD, xUpdate_KNX := i = 81, typDPT := typDPT);
(* LC601_OP *)
(* LC601_CMD *)
M2_207_5N301_LC601_OP(bPortKNX := 2, dwIndex_DPT := 207, rValue_IN := STLV80_563.STLV80_A_563_5N301.LC601_OP, xUpdate_KNX := i = 82, typDPT := typDPT);
M2_208_5N301_LC601_CMD(bPortKNX := 2, dwIndex_DPT := 208, xSwitch_IN := STLV80_563.STLV80_A_563_5N301.LC601_CMD, xUpdate_KNX := i = 83, typDPT := typDPT);
(* RT601_SP *)
(* RT601_SP Feedback *)
M2_209_5N301_RT601_SP(bPortKNX := 2, dwIndex_DPT := 209, rValue_IN := STLV80_563.STLV80_A_563_5N301.RT601_SP_D, xUpdate_KNX := NOT STLV80_563.STLV80_A_563_5N301.RB601_HVAC, typDPT := typDPT);
M2_210_5N301_RT601_SP_FB(bPortKNX := 2, dwIndex_DPT := 210, typDPT := typDPT);
STLV80_563.STLV80_A_563_5N301.RT601_SP_IN := M2_210_5N301_RT601_SP_FB.rValue_OUT;
(* Rom 5N302 *)
(* RB601_V *)
(* RB601_HVAC *)
M2_211_5N302_RB601_V(bPortKNX := 2, dwIndex_DPT := 211, typDPT := typDPT);
STLV80_563.STLV80_A_563_5N302.RB601_V := M2_211_5N302_RB601_V.xSwitch_OUT;
M2_212_5N302_RB601_HVAC(bPortKNX := 2, dwIndex_DPT := 212, typDPT := typDPT);
STLV80_563.STLV80_A_563_5N302.RB601_HVAC := M2_212_5N302_RB601_HVAC.xSwitch_OUT;
(* RT601_CT *)
(* RY601_CV *)
M2_213_5N302_RT601_CT(bPortKNX := 2, dwIndex_DPT := 213, typDPT := typDPT);
STLV80_563.STLV80_A_563_5N302.RT601_CT := M2_213_5N302_RT601_CT.rValue_OUT;
M2_214_5N302_RY601_CV(bPortKNX := 2, dwIndex_DPT := 214, typDPT := typDPT);
STLV80_563.STLV80_A_563_5N302.RY601_CV := M2_214_5N302_RY601_CV.rValue_OUT;
(* LH601_OP *)
(* LH601_CMD *)
M2_215_5N302_LH601_OP(bPortKNX := 2, dwIndex_DPT := 215, rValue_IN := STLV80_563.STLV80_A_563_5N302.LH601_OP, xUpdate_KNX := i = 84, typDPT := typDPT);
M2_216_5N302_LH601_CMD(bPortKNX := 2, dwIndex_DPT := 216, xSwitch_IN := STLV80_563.STLV80_A_563_5N302.LH601_CMD, xUpdate_KNX := i = 85, typDPT := typDPT);
(* LC601_OP *)
(* LC601_CMD *)
M2_217_5N302_LC601_OP(bPortKNX := 2, dwIndex_DPT := 217, rValue_IN := STLV80_563.STLV80_A_563_5N302.LC601_OP, xUpdate_KNX := i = 86, typDPT := typDPT);
M2_218_5N302_LC601_CMD(bPortKNX := 2, dwIndex_DPT := 218, xSwitch_IN := STLV80_563.STLV80_A_563_5N302.LC601_CMD, xUpdate_KNX := i = 87, typDPT := typDPT);
(* RT601_SP *)
(* RT601_SP Feedback *)
M2_219_5N302_RT601_SP(bPortKNX := 2, dwIndex_DPT := 219, rValue_IN := STLV80_563.STLV80_A_563_5N302.RT601_SP_D, xUpdate_KNX := NOT STLV80_563.STLV80_A_563_5N302.RB601_HVAC, typDPT := typDPT);
M2_220_5N302_RT601_SP_FB(bPortKNX := 2, dwIndex_DPT := 220, typDPT := typDPT);
STLV80_563.STLV80_A_563_5N302.RT601_SP_IN := M2_220_5N302_RT601_SP_FB.rValue_OUT;
(* Rom 5O302 *)
(* RB601_V *)
(* RB601_HVAC *)
M2_221_5O302_RB601_V(bPortKNX := 2, dwIndex_DPT := 221, typDPT := typDPT);
STLV80_563.STLV80_A_563_5O302.RB601_V := M2_221_5O302_RB601_V.xSwitch_OUT;
M2_222_5O302_RB601_HVAC(bPortKNX := 2, dwIndex_DPT := 222, typDPT := typDPT);
STLV80_563.STLV80_A_563_5O302.RB601_HVAC := M2_222_5O302_RB601_HVAC.xSwitch_OUT;
(* RT601_CT *)
(* RY601_CV *)
M2_223_5O302_RT601_CT(bPortKNX := 2, dwIndex_DPT := 223, typDPT := typDPT);
STLV80_563.STLV80_A_563_5O302.RT601_CT := M2_223_5O302_RT601_CT.rValue_OUT;
M2_224_5O302_RY601_CV(bPortKNX := 2, dwIndex_DPT := 224, typDPT := typDPT);
STLV80_563.STLV80_A_563_5O302.RY601_CV := M2_224_5O302_RY601_CV.rValue_OUT;
(* LH601_OP *)
(* LH601_CMD *)
M2_225_5O302_LH601_OP(bPortKNX := 2, dwIndex_DPT := 225, rValue_IN := STLV80_563.STLV80_A_563_5O302.LH601_OP, xUpdate_KNX := i = 88, typDPT := typDPT);
M2_226_5O302_LH601_CMD(bPortKNX := 2, dwIndex_DPT := 226, xSwitch_IN := STLV80_563.STLV80_A_563_5O302.LH601_CMD, xUpdate_KNX := i = 89, typDPT := typDPT);
(* LC601_OP *)
(* LC601_CMD *)
M2_227_5O302_LC601_OP(bPortKNX := 2, dwIndex_DPT := 227, rValue_IN := STLV80_563.STLV80_A_563_5O302.LC601_OP, xUpdate_KNX := i = 90, typDPT := typDPT);
M2_228_5O302_LC601_CMD(bPortKNX := 2, dwIndex_DPT := 228, xSwitch_IN := STLV80_563.STLV80_A_563_5O302.LC601_CMD, xUpdate_KNX := i = 91, typDPT := typDPT);
(* RT601_SP *)
(* RT601_SP Feedback *)
M2_229_5O302_RT601_SP(bPortKNX := 2, dwIndex_DPT := 229, rValue_IN := STLV80_563.STLV80_A_563_5O302.RT601_SP_D, xUpdate_KNX := NOT STLV80_563.STLV80_A_563_5O302.RB601_HVAC, typDPT := typDPT);
M2_230_5O302_RT601_SP_FB(bPortKNX := 2, dwIndex_DPT := 230, typDPT := typDPT);
STLV80_563.STLV80_A_563_5O302.RT601_SP_IN := M2_230_5O302_RT601_SP_FB.rValue_OUT;
(* Rom 5O201 *)
(* RB601_V *)
(* RB601_HVAC *)
M2_231_5O201_RB601_V(bPortKNX := 2, dwIndex_DPT := 231, typDPT := typDPT);
STLV80_563.STLV80_A_563_5O201.RB601_V := M2_231_5O201_RB601_V.xSwitch_OUT;
M2_232_5O201_RB601_HVAC(bPortKNX := 2, dwIndex_DPT := 232, typDPT := typDPT);
STLV80_563.STLV80_A_563_5O201.RB601_HVAC := M2_232_5O201_RB601_HVAC.xSwitch_OUT;
(* RT601_CT *)
(* RY601_CV *)
M2_233_5O201_RT601_CT(bPortKNX := 2, dwIndex_DPT := 233, typDPT := typDPT);
STLV80_563.STLV80_A_563_5O201.RT601_CT := M2_233_5O201_RT601_CT.rValue_OUT;
M2_234_5O201_RY601_CV(bPortKNX := 2, dwIndex_DPT := 234, typDPT := typDPT);
STLV80_563.STLV80_A_563_5O201.RY601_CV := M2_234_5O201_RY601_CV.rValue_OUT;
(* LH601_OP *)
(* LH601_CMD *)
M2_235_5O201_LH601_OP(bPortKNX := 2, dwIndex_DPT := 235, rValue_IN := STLV80_563.STLV80_A_563_5O201.LH601_OP, xUpdate_KNX := i = 92, typDPT := typDPT);
M2_236_5O201_LH601_CMD(bPortKNX := 2, dwIndex_DPT := 236, xSwitch_IN := STLV80_563.STLV80_A_563_5O201.LH601_CMD, xUpdate_KNX := i = 93, typDPT := typDPT);
(* LC601_OP *)
(* LC601_CMD *)
M2_237_5O201_LC601_OP(bPortKNX := 2, dwIndex_DPT := 237, rValue_IN := STLV80_563.STLV80_A_563_5O201.LC601_OP, xUpdate_KNX := i = 94, typDPT := typDPT);
M2_238_5O201_LC601_CMD(bPortKNX := 2, dwIndex_DPT := 238, xSwitch_IN := STLV80_563.STLV80_A_563_5O201.LC601_CMD, xUpdate_KNX := i = 95, typDPT := typDPT);
(* RT601_SP *)
(* RT601_SP Feedback *)
M2_239_5O201_RT601_SP(bPortKNX := 2, dwIndex_DPT := 239, rValue_IN := STLV80_563.STLV80_A_563_5O201.RT601_SP_D, xUpdate_KNX := NOT STLV80_563.STLV80_A_563_5O201.RB601_HVAC, typDPT := typDPT);
M2_240_5O201_RT601_SP_FB(bPortKNX := 2, dwIndex_DPT := 240, typDPT := typDPT);
STLV80_563.STLV80_A_563_5O201.RT601_SP_IN := M2_240_5O201_RT601_SP_FB.rValue_OUT;
(* Rom 5O202 *)
(* RB601_V *)
(* RB601_HVAC *)
M2_241_5O202_RB601_V(bPortKNX := 2, dwIndex_DPT := 241, typDPT := typDPT);
STLV80_563.STLV80_A_563_5O202.RB601_V := M2_241_5O202_RB601_V.xSwitch_OUT;
M2_242_5O202_RB601_HVAC(bPortKNX := 2, dwIndex_DPT := 242, typDPT := typDPT);
STLV80_563.STLV80_A_563_5O202.RB601_HVAC := M2_242_5O202_RB601_HVAC.xSwitch_OUT;
(* RT601_CT *)
(* RY601_CV *)
M2_243_5O202_RT601_CT(bPortKNX := 2, dwIndex_DPT := 243, typDPT := typDPT);
STLV80_563.STLV80_A_563_5O202.RT601_CT := M2_243_5O202_RT601_CT.rValue_OUT;
M2_244_5O202_RY601_CV(bPortKNX := 2, dwIndex_DPT := 244, typDPT := typDPT);
STLV80_563.STLV80_A_563_5O202.RY601_CV := M2_244_5O202_RY601_CV.rValue_OUT;
(* LH601_OP *)
(* LH601_CMD *)
M2_245_5O202_LH601_OP(bPortKNX := 2, dwIndex_DPT := 245, rValue_IN := STLV80_563.STLV80_A_563_5O202.LH601_OP, xUpdate_KNX := i = 96, typDPT := typDPT);
M2_246_5O202_LH601_CMD(bPortKNX := 2, dwIndex_DPT := 246, xSwitch_IN := STLV80_563.STLV80_A_563_5O202.LH601_CMD, xUpdate_KNX := i = 97, typDPT := typDPT);
(* LC601_OP *)
(* LC601_CMD *)
M2_247_5O202_LC601_OP(bPortKNX := 2, dwIndex_DPT := 247, rValue_IN := STLV80_563.STLV80_A_563_5O202.LC601_OP, xUpdate_KNX := i = 98, typDPT := typDPT);
M2_248_5O202_LC601_CMD(bPortKNX := 2, dwIndex_DPT := 248, xSwitch_IN := STLV80_563.STLV80_A_563_5O202.LC601_CMD, xUpdate_KNX := i = 99, typDPT := typDPT);
(* RT601_SP *)
(* RT601_SP Feedback *)
M2_249_5O202_RT601_SP(bPortKNX := 2, dwIndex_DPT := 249, rValue_IN := STLV80_563.STLV80_A_563_5O202.RT601_SP_D, xUpdate_KNX := NOT STLV80_563.STLV80_A_563_5O202.RB601_HVAC, typDPT := typDPT);
M2_250_5O202_RT601_SP_FB(bPortKNX := 2, dwIndex_DPT := 250, typDPT := typDPT);
STLV80_563.STLV80_A_563_5O202.RT601_SP_IN := M2_250_5O202_RT601_SP_FB.rValue_OUT;
END_PROGRAM

PROGRAM PRG_563_KNX_3
  VAR
    i : INT := 0;  (* Felles *)
    Interval : OSCAT_BASIC.CLK_PRG;
    typDPT : typDPT;
    KNX_master_3 : WagoAppKNX.FbKNX_Master;  (* Master *)
    M3_001_5O301_RB601_V : fbDPT_Switch_pro;  (* 5O301 *)
    M3_002_5O301_RB601_HVAC : fbDPT_Switch_pro;
    M3_003_5O301_RT601_CT : fbDPT_Value_Temp_pro;
    M3_004_5O301_RY601_CV : fbDPT_Value_AirQuality_pro;
    M3_005_5O301_LH601_OP : fbDPT_Scaling_pro;
    M3_006_5O301_LH601_CMD : fbDPT_Switch_pro;
    M3_007_5O301_LC601_OP : fbDPT_Scaling_pro;
    M3_008_5O301_LC601_CMD : fbDPT_Switch_pro;
    M3_009_5O301_RT601_SP : fbDPT_Value_Temp_pro;
    M3_010_5O301_RT601_SP_FB : fbDPT_Value_Temp_pro;
    M3_011_5P302_RB601_V : fbDPT_Switch_pro;  (* 5P302 *)
    M3_012_5P302_RB601_HVAC : fbDPT_Switch_pro;
    M3_013_5P302_RT601_CT : fbDPT_Value_Temp_pro;
    M3_014_5P302_RY601_CV : fbDPT_Value_AirQuality_pro;
    M3_015_5P302_LH601_OP : fbDPT_Scaling_pro;
    M3_016_5P302_LH601_CMD : fbDPT_Switch_pro;
    M3_017_5P302_LC601_OP : fbDPT_Scaling_pro;
    M3_018_5P302_LC601_CMD : fbDPT_Switch_pro;
    M3_019_5P302_RT601_SP : fbDPT_Value_Temp_pro;
    M3_020_5P302_RT601_SP_FB : fbDPT_Value_Temp_pro;
    M3_021_5P201_RB601_V : fbDPT_Switch_pro;  (* 5P201 *)
    M3_022_5P201_RB601_HVAC : fbDPT_Switch_pro;
    M3_023_5P201_RT601_CT : fbDPT_Value_Temp_pro;
    M3_024_5P201_RY601_CV : fbDPT_Value_AirQuality_pro;
    M3_025_5P201_LH601_OP : fbDPT_Scaling_pro;
    M3_026_5P201_LH601_CMD : fbDPT_Switch_pro;
    M3_027_5P201_LC601_OP : fbDPT_Scaling_pro;
    M3_028_5P201_LC601_CMD : fbDPT_Switch_pro;
    M3_029_5P201_RT601_SP : fbDPT_Value_Temp_pro;
    M3_030_5P201_RT601_SP_FB : fbDPT_Value_Temp_pro;
    M3_031_5P202_RB601_V : fbDPT_Switch_pro;  (* 5P202 *)
    M3_032_5P202_RB601_HVAC : fbDPT_Switch_pro;
    M3_033_5P202_RT601_CT : fbDPT_Value_Temp_pro;
    M3_034_5P202_RY601_CV : fbDPT_Value_AirQuality_pro;
    M3_035_5P202_LH601_OP : fbDPT_Scaling_pro;
    M3_036_5P202_LH601_CMD : fbDPT_Switch_pro;
    M3_037_5P202_LC601_OP : fbDPT_Scaling_pro;
    M3_038_5P202_LC601_CMD : fbDPT_Switch_pro;
    M3_039_5P202_RT601_SP : fbDPT_Value_Temp_pro;
    M3_040_5P202_RT601_SP_FB : fbDPT_Value_Temp_pro;
    M3_041_5Q301_RB601_V : fbDPT_Switch_pro;  (* 5Q301 *)
    M3_042_5Q301_RB601_HVAC : fbDPT_Switch_pro;
    M3_043_5Q301_RT601_CT : fbDPT_Value_Temp_pro;
    M3_044_5Q301_RY601_CV : fbDPT_Value_AirQuality_pro;
    M3_045_5Q301_LH601_OP : fbDPT_Scaling_pro;
    M3_046_5Q301_LH601_CMD : fbDPT_Switch_pro;
    M3_047_5Q301_LC601_OP : fbDPT_Scaling_pro;
    M3_048_5Q301_LC601_CMD : fbDPT_Switch_pro;
    M3_049_5Q301_RT601_SP : fbDPT_Value_Temp_pro;
    M3_050_5Q301_RT601_SP_FB : fbDPT_Value_Temp_pro;
    M3_051_5Q302_RB601_V : fbDPT_Switch_pro;  (* 5Q302 *)
    M3_052_5Q302_RB601_HVAC : fbDPT_Switch_pro;
    M3_053_5Q302_RT601_CT : fbDPT_Value_Temp_pro;
    M3_054_5Q302_RY601_CV : fbDPT_Value_AirQuality_pro;
    M3_055_5Q302_LH601_OP : fbDPT_Scaling_pro;
    M3_056_5Q302_LH601_CMD : fbDPT_Switch_pro;
    M3_057_5Q302_LC601_OP : fbDPT_Scaling_pro;
    M3_058_5Q302_LC601_CMD : fbDPT_Switch_pro;
    M3_059_5Q302_RT601_SP : fbDPT_Value_Temp_pro;
    M3_060_5Q302_RT601_SP_FB : fbDPT_Value_Temp_pro;
  END_VAR

(* CFC diagram, written out as Structured Text *)
(* KNX Master *)
KNX_master_3(I_Port := IoConfig_Globals.KNX_EIB_TP1_Interface_2, bPortKNX := 3);
STLV80_563.STLV80_A_563_KNX_Card_3_Status := KNX_master_3.sStatus = 'OK';
(* Rom 5O301 *)
(* RB601_V *)
(* RB601_HVAC *)
M3_001_5O301_RB601_V(bPortKNX := 3, dwIndex_DPT := 1, typDPT := typDPT);
STLV80_563.STLV80_A_563_5O301.RB601_V := M3_001_5O301_RB601_V.xSwitch_OUT;
M3_002_5O301_RB601_HVAC(bPortKNX := 3, dwIndex_DPT := 2, typDPT := typDPT);
STLV80_563.STLV80_A_563_5O301.RB601_HVAC := M3_002_5O301_RB601_HVAC.xSwitch_OUT;
(* RT601_CT *)
(* RY601_CV *)
M3_003_5O301_RT601_CT(bPortKNX := 3, dwIndex_DPT := 3, typDPT := typDPT);
STLV80_563.STLV80_A_563_5O301.RT601_CT := M3_003_5O301_RT601_CT.rValue_OUT;
M3_004_5O301_RY601_CV(bPortKNX := 3, dwIndex_DPT := 4, typDPT := typDPT);
STLV80_563.STLV80_A_563_5O301.RY601_CV := M3_004_5O301_RY601_CV.rValue_OUT;
(* LH601_OP *)
(* LH601_CMD *)
M3_005_5O301_LH601_OP(bPortKNX := 3, dwIndex_DPT := 5, rValue_IN := STLV80_563.STLV80_A_563_5O301.LH601_OP, xUpdate_KNX := i = 0, typDPT := typDPT);
M3_006_5O301_LH601_CMD(bPortKNX := 3, dwIndex_DPT := 6, xSwitch_IN := STLV80_563.STLV80_A_563_5O301.LH601_CMD, xUpdate_KNX := i = 1, typDPT := typDPT);
(* LC601_OP *)
(* LC601_CMD *)
M3_007_5O301_LC601_OP(bPortKNX := 3, dwIndex_DPT := 7, rValue_IN := STLV80_563.STLV80_A_563_5O301.LC601_OP, xUpdate_KNX := i = 2, typDPT := typDPT);
M3_008_5O301_LC601_CMD(bPortKNX := 3, dwIndex_DPT := 8, xSwitch_IN := STLV80_563.STLV80_A_563_5O301.LC601_CMD, xUpdate_KNX := i = 3, typDPT := typDPT);
(* RT601_SP *)
(* RT601_SP Feedback *)
M3_009_5O301_RT601_SP(bPortKNX := 3, dwIndex_DPT := 9, rValue_IN := STLV80_563.STLV80_A_563_5O301.RT601_SP_D, xUpdate_KNX := NOT STLV80_563.STLV80_A_563_5O301.RB601_HVAC, typDPT := typDPT);
M3_010_5O301_RT601_SP_FB(bPortKNX := 3, dwIndex_DPT := 10, typDPT := typDPT);
STLV80_563.STLV80_A_563_5O301.RT601_SP_IN := M3_010_5O301_RT601_SP_FB.rValue_OUT;
(* Rom 5P302 *)
(* RB601_V *)
(* RB601_HVAC *)
M3_011_5P302_RB601_V(bPortKNX := 3, dwIndex_DPT := 11, typDPT := typDPT);
STLV80_563.STLV80_A_563_5P302.RB601_V := M3_011_5P302_RB601_V.xSwitch_OUT;
M3_012_5P302_RB601_HVAC(bPortKNX := 3, dwIndex_DPT := 12, typDPT := typDPT);
STLV80_563.STLV80_A_563_5P302.RB601_HVAC := M3_012_5P302_RB601_HVAC.xSwitch_OUT;
(* RT601_CT *)
(* RY601_CV *)
M3_013_5P302_RT601_CT(bPortKNX := 3, dwIndex_DPT := 13, typDPT := typDPT);
STLV80_563.STLV80_A_563_5P302.RT601_CT := M3_013_5P302_RT601_CT.rValue_OUT;
M3_014_5P302_RY601_CV(bPortKNX := 3, dwIndex_DPT := 14, typDPT := typDPT);
STLV80_563.STLV80_A_563_5P302.RY601_CV := M3_014_5P302_RY601_CV.rValue_OUT;
(* LH601_OP *)
(* LH601_CMD *)
M3_015_5P302_LH601_OP(bPortKNX := 3, dwIndex_DPT := 15, rValue_IN := STLV80_563.STLV80_A_563_5P302.LH601_OP, xUpdate_KNX := i = 4, typDPT := typDPT);
M3_016_5P302_LH601_CMD(bPortKNX := 3, dwIndex_DPT := 16, xSwitch_IN := STLV80_563.STLV80_A_563_5P302.LH601_CMD, xUpdate_KNX := i = 5, typDPT := typDPT);
(* LC601_OP *)
(* LC601_CMD *)
M3_017_5P302_LC601_OP(bPortKNX := 3, dwIndex_DPT := 17, rValue_IN := STLV80_563.STLV80_A_563_5P302.LC601_OP, xUpdate_KNX := i = 6, typDPT := typDPT);
M3_018_5P302_LC601_CMD(bPortKNX := 3, dwIndex_DPT := 18, xSwitch_IN := STLV80_563.STLV80_A_563_5P302.LC601_CMD, xUpdate_KNX := i = 7, typDPT := typDPT);
(* RT601_SP *)
(* RT601_SP Feedback *)
M3_019_5P302_RT601_SP(bPortKNX := 3, dwIndex_DPT := 19, rValue_IN := STLV80_563.STLV80_A_563_5P302.RT601_SP_D, xUpdate_KNX := NOT STLV80_563.STLV80_A_563_5P302.RB601_HVAC, typDPT := typDPT);
M3_020_5P302_RT601_SP_FB(bPortKNX := 3, dwIndex_DPT := 20, typDPT := typDPT);
STLV80_563.STLV80_A_563_5P302.RT601_SP_IN := M3_020_5P302_RT601_SP_FB.rValue_OUT;
(* Rom 5P201 *)
(* RB601_V *)
(* RB601_HVAC *)
M3_021_5P201_RB601_V(bPortKNX := 3, dwIndex_DPT := 21, typDPT := typDPT);
STLV80_563.STLV80_A_563_5P201.RB601_V := M3_021_5P201_RB601_V.xSwitch_OUT;
M3_022_5P201_RB601_HVAC(bPortKNX := 3, dwIndex_DPT := 22, typDPT := typDPT);
STLV80_563.STLV80_A_563_5P201.RB601_HVAC := M3_022_5P201_RB601_HVAC.xSwitch_OUT;
(* RT601_CT *)
(* RY601_CV *)
M3_023_5P201_RT601_CT(bPortKNX := 3, dwIndex_DPT := 23, typDPT := typDPT);
STLV80_563.STLV80_A_563_5P201.RT601_CT := M3_023_5P201_RT601_CT.rValue_OUT;
M3_024_5P201_RY601_CV(bPortKNX := 3, dwIndex_DPT := 24, typDPT := typDPT);
STLV80_563.STLV80_A_563_5P201.RY601_CV := M3_024_5P201_RY601_CV.rValue_OUT;
(* LH601_OP *)
(* LH601_CMD *)
M3_025_5P201_LH601_OP(bPortKNX := 3, dwIndex_DPT := 25, rValue_IN := STLV80_563.STLV80_A_563_5P201.LH601_OP, xUpdate_KNX := i = 8, typDPT := typDPT);
M3_026_5P201_LH601_CMD(bPortKNX := 3, dwIndex_DPT := 26, xSwitch_IN := STLV80_563.STLV80_A_563_5P201.LH601_CMD, xUpdate_KNX := i = 9, typDPT := typDPT);
(* LC601_OP *)
(* LC601_CMD *)
M3_027_5P201_LC601_OP(bPortKNX := 3, dwIndex_DPT := 27, rValue_IN := STLV80_563.STLV80_A_563_5P201.LC601_OP, xUpdate_KNX := i = 10, typDPT := typDPT);
M3_028_5P201_LC601_CMD(bPortKNX := 3, dwIndex_DPT := 28, xSwitch_IN := STLV80_563.STLV80_A_563_5P201.LC601_CMD, xUpdate_KNX := i = 11, typDPT := typDPT);
(* RT601_SP *)
(* RT601_SP Feedback *)
M3_029_5P201_RT601_SP(bPortKNX := 3, dwIndex_DPT := 29, rValue_IN := STLV80_563.STLV80_A_563_5P201.RT601_SP_D, xUpdate_KNX := NOT STLV80_563.STLV80_A_563_5P201.RB601_HVAC, typDPT := typDPT);
M3_030_5P201_RT601_SP_FB(bPortKNX := 3, dwIndex_DPT := 30, typDPT := typDPT);
STLV80_563.STLV80_A_563_5P201.RT601_SP_IN := M3_030_5P201_RT601_SP_FB.rValue_OUT;
(* Rom 5P202 *)
(* RB601_V *)
(* RB601_HVAC *)
M3_031_5P202_RB601_V(bPortKNX := 3, dwIndex_DPT := 31, typDPT := typDPT);
STLV80_563.STLV80_A_563_5P202.RB601_V := M3_031_5P202_RB601_V.xSwitch_OUT;
M3_032_5P202_RB601_HVAC(bPortKNX := 3, dwIndex_DPT := 32, typDPT := typDPT);
STLV80_563.STLV80_A_563_5P202.RB601_HVAC := M3_032_5P202_RB601_HVAC.xSwitch_OUT;
(* RT601_CT *)
(* RY601_CV *)
M3_033_5P202_RT601_CT(bPortKNX := 3, dwIndex_DPT := 33, typDPT := typDPT);
STLV80_563.STLV80_A_563_5P202.RT601_CT := M3_033_5P202_RT601_CT.rValue_OUT;
M3_034_5P202_RY601_CV(bPortKNX := 3, dwIndex_DPT := 34, typDPT := typDPT);
STLV80_563.STLV80_A_563_5P202.RY601_CV := M3_034_5P202_RY601_CV.rValue_OUT;
(* LH601_OP *)
(* LH601_CMD *)
M3_035_5P202_LH601_OP(bPortKNX := 3, dwIndex_DPT := 35, rValue_IN := STLV80_563.STLV80_A_563_5P202.LH601_OP, xUpdate_KNX := i = 12, typDPT := typDPT);
M3_036_5P202_LH601_CMD(bPortKNX := 3, dwIndex_DPT := 36, xSwitch_IN := STLV80_563.STLV80_A_563_5P202.LH601_CMD, xUpdate_KNX := i = 13, typDPT := typDPT);
(* LC601_OP *)
(* LC601_CMD *)
M3_037_5P202_LC601_OP(bPortKNX := 3, dwIndex_DPT := 37, rValue_IN := STLV80_563.STLV80_A_563_5P202.LC601_OP, xUpdate_KNX := i = 14, typDPT := typDPT);
M3_038_5P202_LC601_CMD(bPortKNX := 3, dwIndex_DPT := 38, xSwitch_IN := STLV80_563.STLV80_A_563_5P202.LC601_CMD, xUpdate_KNX := i = 15, typDPT := typDPT);
(* RT601_SP *)
(* RT601_SP Feedback *)
M3_039_5P202_RT601_SP(bPortKNX := 3, dwIndex_DPT := 39, rValue_IN := STLV80_563.STLV80_A_563_5P202.RT601_SP_D, xUpdate_KNX := NOT STLV80_563.STLV80_A_563_5P202.RB601_HVAC, typDPT := typDPT);
M3_040_5P202_RT601_SP_FB(bPortKNX := 3, dwIndex_DPT := 40, typDPT := typDPT);
STLV80_563.STLV80_A_563_5P202.RT601_SP_IN := M3_040_5P202_RT601_SP_FB.rValue_OUT;
(* Rom 5Q301 *)
(* RB601_V *)
(* RB601_HVAC *)
M3_041_5Q301_RB601_V(bPortKNX := 3, dwIndex_DPT := 41, typDPT := typDPT);
STLV80_563.STLV80_A_563_5Q301.RB601_V := M3_041_5Q301_RB601_V.xSwitch_OUT;
M3_042_5Q301_RB601_HVAC(bPortKNX := 3, dwIndex_DPT := 42, typDPT := typDPT);
STLV80_563.STLV80_A_563_5Q301.RB601_HVAC := M3_042_5Q301_RB601_HVAC.xSwitch_OUT;
(* RT601_CT *)
(* RY601_CV *)
M3_043_5Q301_RT601_CT(bPortKNX := 3, dwIndex_DPT := 43, typDPT := typDPT);
STLV80_563.STLV80_A_563_5Q301.RT601_CT := M3_043_5Q301_RT601_CT.rValue_OUT;
M3_044_5Q301_RY601_CV(bPortKNX := 3, dwIndex_DPT := 44, typDPT := typDPT);
STLV80_563.STLV80_A_563_5Q301.RY601_CV := M3_044_5Q301_RY601_CV.rValue_OUT;
(* LH601_OP *)
(* LH601_CMD *)
M3_045_5Q301_LH601_OP(bPortKNX := 3, dwIndex_DPT := 45, rValue_IN := STLV80_563.STLV80_A_563_5Q301.LH601_OP, xUpdate_KNX := i = 16, typDPT := typDPT);
M3_046_5Q301_LH601_CMD(bPortKNX := 3, dwIndex_DPT := 46, xSwitch_IN := STLV80_563.STLV80_A_563_5Q301.LH601_CMD, xUpdate_KNX := i = 17, typDPT := typDPT);
(* LC601_OP *)
(* LC601_CMD *)
M3_047_5Q301_LC601_OP(bPortKNX := 3, dwIndex_DPT := 47, rValue_IN := STLV80_563.STLV80_A_563_5Q301.LC601_OP, xUpdate_KNX := i = 18, typDPT := typDPT);
M3_048_5Q301_LC601_CMD(bPortKNX := 3, dwIndex_DPT := 48, xSwitch_IN := STLV80_563.STLV80_A_563_5Q301.LC601_CMD, xUpdate_KNX := i = 19, typDPT := typDPT);
(* RT601_SP *)
(* RT601_SP Feedback *)
M3_049_5Q301_RT601_SP(bPortKNX := 3, dwIndex_DPT := 49, rValue_IN := STLV80_563.STLV80_A_563_5Q301.RT601_SP_D, xUpdate_KNX := NOT STLV80_563.STLV80_A_563_5Q301.RB601_HVAC, typDPT := typDPT);
M3_050_5Q301_RT601_SP_FB(bPortKNX := 3, dwIndex_DPT := 50, typDPT := typDPT);
STLV80_563.STLV80_A_563_5Q301.RT601_SP_IN := M3_050_5Q301_RT601_SP_FB.rValue_OUT;
(* Rom 5Q302 *)
(* RB601_V *)
(* RB601_HVAC *)
M3_051_5Q302_RB601_V(bPortKNX := 3, dwIndex_DPT := 51, typDPT := typDPT);
STLV80_563.STLV80_A_563_5Q302.RB601_V := M3_051_5Q302_RB601_V.xSwitch_OUT;
M3_052_5Q302_RB601_HVAC(bPortKNX := 3, dwIndex_DPT := 52, typDPT := typDPT);
STLV80_563.STLV80_A_563_5Q302.RB601_HVAC := M3_052_5Q302_RB601_HVAC.xSwitch_OUT;
(* RT601_CT *)
(* RY601_CV *)
M3_053_5Q302_RT601_CT(bPortKNX := 3, dwIndex_DPT := 53, typDPT := typDPT);
STLV80_563.STLV80_A_563_5Q302.RT601_CT := M3_053_5Q302_RT601_CT.rValue_OUT;
M3_054_5Q302_RY601_CV(bPortKNX := 3, dwIndex_DPT := 54, typDPT := typDPT);
STLV80_563.STLV80_A_563_5Q302.RY601_CV := M3_054_5Q302_RY601_CV.rValue_OUT;
(* LH601_OP *)
(* LH601_CMD *)
M3_055_5Q302_LH601_OP(bPortKNX := 3, dwIndex_DPT := 55, rValue_IN := STLV80_563.STLV80_A_563_5Q302.LH601_OP, xUpdate_KNX := i = 20, typDPT := typDPT);
M3_056_5Q302_LH601_CMD(bPortKNX := 3, dwIndex_DPT := 56, xSwitch_IN := STLV80_563.STLV80_A_563_5Q302.LH601_CMD, xUpdate_KNX := i = 21, typDPT := typDPT);
(* LC601_OP *)
(* LC601_CMD *)
M3_057_5Q302_LC601_OP(bPortKNX := 3, dwIndex_DPT := 57, rValue_IN := STLV80_563.STLV80_A_563_5Q302.LC601_OP, xUpdate_KNX := i = 22, typDPT := typDPT);
M3_058_5Q302_LC601_CMD(bPortKNX := 3, dwIndex_DPT := 58, xSwitch_IN := STLV80_563.STLV80_A_563_5Q302.LC601_CMD, xUpdate_KNX := i = 23, typDPT := typDPT);
(* RT601_SP *)
(* RT601_SP Feedback *)
M3_059_5Q302_RT601_SP(bPortKNX := 3, dwIndex_DPT := 59, rValue_IN := STLV80_563.STLV80_A_563_5Q302.RT601_SP_D, xUpdate_KNX := NOT STLV80_563.STLV80_A_563_5Q302.RB601_HVAC, typDPT := typDPT);
M3_060_5Q302_RT601_SP_FB(bPortKNX := 3, dwIndex_DPT := 60, typDPT := typDPT);
STLV80_563.STLV80_A_563_5Q302.RT601_SP_IN := M3_060_5Q302_RT601_SP_FB.rValue_OUT;
END_PROGRAM
